{attribute 'GeneratedUsingTerminal: EL6201-0000-0017'}
{attribute addProperty BoxType "EL6201-0000-0017"}
{attribute addProperty Id "Slave_30A_DI0BOOL1Slave_30A_DI1BOOL1Slave_30A_DI2BOOL1Slave_30A_DI3BOOL1Slave_30B_DI0BOOL1Slave_30B_DI1BOOL1Slave_30B_DI2BOOL1Slave_30B_DI3BOOL1"}
{attribute addProperty CRC "429673898"}
{attribute addProperty Size "8"}
TYPE Slave_30_Inputs_199C4DAA :
STRUCT
	{attribute addProperty Name "Slave_30A_DI0"}
	Slave_30A_DI0 : BOOL;
	{attribute addProperty Name "Slave_30A_DI1"}
	Slave_30A_DI1 : BOOL;
	{attribute addProperty Name "Slave_30A_DI2"}
	Slave_30A_DI2 : BOOL;
	{attribute addProperty Name "Slave_30A_DI3"}
	Slave_30A_DI3 : BOOL;
	{attribute addProperty Name "Slave_30B_DI0"}
	Slave_30B_DI0 : BOOL;
	{attribute addProperty Name "Slave_30B_DI1"}
	Slave_30B_DI1 : BOOL;
	{attribute addProperty Name "Slave_30B_DI2"}
	Slave_30B_DI2 : BOOL;
	{attribute addProperty Name "Slave_30B_DI3"}
	Slave_30B_DI3 : BOOL;
END_STRUCT
END_TYPE

(* stored: Version 1.2.0.0, ProductVersion 3.1.4024.9
   DUT Slave_30_Inputs_199C4DAA: Id {44e1c0a7-f2de-4171-9485-e794ae6ac07c} *)
